// TwinCAT 3 PLC project Untitled1
// ProgramVersion: 3.1.4024.0
// libraries:
//   Tc2_Standard, * (Beckhoff Automation GmbH)
//   Tc2_System, * (Beckhoff Automation GmbH)
//   Tc3_Module, * (Beckhoff Automation GmbH)
// project tree:
//   DUTs/ KOMANDA.TcDUT (not stored), POZAYZ.TcDUT (not stored), POZICIJA.TcDUT (not stored), Valj.TcDUT (not stored)
//   GVLs/ AUTO.TcGVL, GVL.TcGVL (not stored)
//   / PlcTask.TcTTO (not stored)
//   POUs/ AutoMove.TcPOU (not stored), Counter.TcPOU (not stored), Init.TcPOU, MAIN.TcPOU (not stored), Motor.TcPOU (not stored), MotorControla.TcPOU, Multiplex.TcPOU (not stored), Automatic.TcPOU, AutoMove2.TcPOU, Test.TcPOU (not stored), TrackingLogic.TcPOU (not stored)
// real-time tasks:
//   TASK PlcTask: cycle T#10ms, priority 20, ADS port 350
// I/O:
//   DEVICE Device 1 (EtherCAT), AmsNetId 5.132.85.185.2.1
//     Term 1 (EK1200) [EK1200-7000 EtherCAT Power supply (1,5A E-Bus)]
//       Term 2 (EL1859) [EL1859 8Ch. Dig. Input 24V, 3ms, 8Ch. Dig. Output 24V, 0.5A]
//       Term 3 (EL1859) [EL1859 8Ch. Dig. Input 24V, 3ms, 8Ch. Dig. Output 24V, 0.5A]
//       Term 4 (EL5152) [EL5152 2Ch. Inc. Encoder]
//       Term 5 (EL9011) [EL9011 End Terminal]
//   DEVICE Device 2 (NOV-DP-RAM)
//   DEVICE Device 5 (CX7000), AmsNetId 5.132.85.185.6.1
//     Term 1 (CX7028) [CX7028-0000-0118]
//       modules: Module 1 (DIO_2x), Module 3 (DIO_2x), Module 5 (DI_2x), Module 7 (DI_2x)
// variable links:
//   Untitled1/Untitled1 Instance <-> Device 1 (EtherCAT)/Term 1 (EK1200)/Term 2 (EL1859)
//     PlcTask Inputs/GVL.KSD <-> Channel 5/Input
//     PlcTask Inputs/GVL.KSI <-> Channel 3/Input
//     PlcTask Inputs/GVL.KSP <-> Channel 7/Input
//     PlcTask Inputs/GVL.KSV <-> Channel 1/Input
//     PlcTask Inputs/GVL.StD <-> Channel 6/Input
//     PlcTask Inputs/GVL.StI <-> Channel 4/Input
//     PlcTask Inputs/GVL.StP <-> Channel 8/Input
//     PlcTask Inputs/GVL.StV <-> Channel 2/Input
//     PlcTask Outputs/GVL.MDP <-> Channel 14/Output
//     PlcTask Outputs/GVL.MDS <-> Channel 13/Output
//     PlcTask Outputs/GVL.MIP <-> Channel 12/Output
//     PlcTask Outputs/GVL.MIS <-> Channel 11/Output
//     PlcTask Outputs/GVL.MPP <-> Channel 16/Output
//     PlcTask Outputs/GVL.MPS <-> Channel 15/Output
//     PlcTask Outputs/GVL.MVP <-> Channel 10/Output
//     PlcTask Outputs/GVL.MVS <-> Channel 9/Output
//   Untitled1/Untitled1 Instance <-> Device 5 (CX7000)/Term 1 (CX7028)
//     PlcTask Inputs/GVL.GreenButton <-> Module 3 (DIO_2x)/DIO_2x Input Channel 2/Input
//     PlcTask Inputs/GVL.LLBButton <-> Module 5 (DI_2x)/DI_2x Input Channel 1/Input
//     PlcTask Inputs/GVL.LRBButton <-> Module 5 (DI_2x)/DI_2x Input Channel 2/Input
//     PlcTask Inputs/GVL.RedButton <-> Module 1 (DIO_2x)/DIO_2x Inputs Channel 1/Input
//     PlcTask Inputs/GVL.ToggleSwitch <-> Module 7 (DI_2x)/DI_2x Inputs Channel 1/Input
//     PlcTask Inputs/GVL.ULBButton <-> Module 1 (DIO_2x)/DIO_2x Inputs Channel 2/Input
//     PlcTask Inputs/GVL.URBButton <-> Module 3 (DIO_2x)/DIO_2x Input Channel 1/Input
//     PlcTask Outputs/GVL.LEDGreen <-> Module 3 (DIO_2x)/DIO_2x Outputs Channel 1/Output
//     PlcTask Outputs/GVL.LEDLBlue <-> Module 3 (DIO_2x)/DIO_2x Outputs Channel 2/Output
//     PlcTask Outputs/GVL.LEDRed <-> Module 1 (DIO_2x)/DIO_2x Outputs Channel 1/Output
//     PlcTask Outputs/GVL.LEDUBlue <-> Module 1 (DIO_2x)/DIO_2x Outputs Channel 2/Output

// ---- GVLs/AUTO.TcGVL
{attribute 'qualified_only'}
VAR_GLOBAL
	Varno :BOOL := FALSE;
	MotorIzbira : INT;
	VrtenjePremik : BOOL;
	VrtenjeSmer : BOOL;
	DvigPremik : BOOL;
	DvigSmer : BOOL;
	IztegPremik : BOOL;
	IztegSmer : BOOL;
	PrijemPremik : BOOL;
	PrijemSmer : BOOL;
	Current: POZICIJA;
	N: INT := 5; //v InstructionSize
	Komande0: ARRAY [0..4] OF POZICIJA := [(A := 0, Y := 0, Z := 0, P:= 0 ), 
		(A := 100, Y := 40, Z := 50, P:= 15 ),
		(A := 80, Y := 20, Z := 30, P:= 0 ),
		(A := 120, Y := 0, Z := 15, P:= 12 ),
		(A := 100, Y := 0, Z := 15, P:= 0 )];
	Status: INT := 0;
	PositionNum: INT := 2; // ne rabi
	ItemNumber : INT := 2; //ne rabi
	StageSelect : INT := 0;
	Recept : INT := 0;
	VRoki : INT := 0;
	Positions: ARRAY [1..11] OF POZAYZ := [
			(A := 30, Y:=60, Z:= 105),
			(A := 30, Y:=60, Z:= 62),
			(A := 30, Y:=60, Z:= 20),
			(A := 60, Y:=60, Z:= 105),
			(A := 60, Y:=60, Z:= 62), // 5
			(A := 50, Y:=60, Z:= 105),
			(A := 50, Y:=60, Z:= 62),
			(A := 37, Y:=60, Z:= 105),
			(A := 40, Y:=45, Z:= 105),
			(A := 43, Y:=60, Z:= 105),
			(A := 33, Y:=0, Z:= 50)]; // 10
	Items: ARRAY [1..5] OF POZAYZ := [
			(A := 5, Y:=60, Z:= 20),
			(A := 5, Y:=60, Z:= 62),
			(A := 5, Y:=60, Z:= 105),
			(A := 50, Y:=60, Z:= 105),
			(A := 50, Y:=60, Z:= 62)];
	StageMax : INT :=10;
	Stages :  ARRAY [1 .. 3] OF ARRAY [1 .. 9] OF KOMANDA :=  [[
		(I := 1, T := 0, P := 16),
		(I := 0, T := 1, P := 0),
		(I := 2, T := 0, P := 16),
		(I := 0, T := 2, P := 0),
		(I := 3, T := 0, P := 16), // 5
		(I := 0, T := 3, P := 0),
		(I := 2, T := 0, P := 16),
		(I := 0, T := 9, P := 0),
		(I := 0, T := 11, P := 0)],
[
		(I := 5, T := 0, P := 16),
		(I := 0, T := 4, P := 0),
		(I := 4, T := 0, P := 16),
		(I := 0, T := 5, P := 0),
		(I := 4, T := 0, P := 16), // 5
		(I := 0, T := 6, P := 0),
		(I := 5, T := 0, P := 16),
		(I := 0, T := 7, P := 0),
		(I := 0, T := 11, P := 0)],
[
		(I := 1, T := 0, P := 16),
		(I := 0, T := 10, P := 0),
		(I := 2, T := 0, P := 16),
		(I := 0, T := 8, P := 0),
		(I := 3, T := 0, P := 16), // 5
		(I := 0, T := 9, P := 0),
		(I := 2, T := 0, P := 16),
		(I := 0, T := 1, P := 0),
		(I := 0, T := 11, P := 0)]];
END_VAR

// ---- POUs/Init.TcPOU
FUNCTION_BLOCK Init
VAR_INPUT
END_VAR
VAR_OUTPUT
END_VAR
VAR
	isInit: BOOL := FALSE;
END_VAR

IF NOT isInit AND GVL.ToggleSwitch = FALSE THEN
	IF NOT GVL.KSV THEN
		AUTO.MotorIzbira := 1;
		AUTO.VrtenjeSmer := TRUE;
		AUTO.VrtenjePremik := TRUE;
	ELSIF NOT GVL.KSD THEN
		AUTO.VrtenjePremik:= FALSE;
		AUTO.MotorIzbira := 2;
		AUTO.DvigSmer := TRUE;
		AUTO.DvigPremik := TRUE;
	ELSIF NOT GVL.KSP THEN
		AUTO.MotorIzbira := 4;
		AUTO.PrijemSmer := TRUE;
		AUTO.PrijemPremik := TRUE;
	ELSE
		AUTO.MotorIzbira := 0;
		AUTO.Current.Y := 0;
		IF GVL.ULBButton = TRUE THEN
			AUTO.Recept := 1;
		ELSIF GVL.URBButton = TRUE THEN
			AUTO.Recept:= 2;
		ELSIF GVL.LLBButton= TRUE THEN
			AUTO.Recept := 3;
		END_IF
		IF AUTO.Recept <> 0 THEN
			AUTO.StageSelect := 1;
			isInit := TRUE;
		END_IF
		
	END_IF
END_IF

END_FUNCTION_BLOCK

// ---- POUs/MotorControla.TcPOU
FUNCTION_BLOCK MotorControla
VAR_INPUT
	Premik: BOOL;
	Smer: BOOL;
	Select: BOOL;
	KS: BOOL;
	Step: BOOL;
	Limes: WORD;
END_VAR
VAR_OUTPUT
	OutPremik: BOOL;
	OutSmer: BOOL;
	Interlock: BOOL;
	Stop: BOOL;
	Position: WORD;
END_VAR
VAR
	R_TRIG_0: R_TRIG;
	Dump: TIME;
	InL: TOF;
	RS_0: RS;

	R_TRIG_1: R_TRIG;
	TON0: TON;
	TON1: TON;
	TON_0: TON;
	Counter_0: Counter;
	F_TRIG_0: F_TRIG;
	InL1: TOF;
	IntL1: BOOL;
	IntL2: BOOL;
	IntL3: BOOL;
END_VAR
//dODAJ COLLISION DETECTION AND AVOIDANCE
//ZRIHTAJ SMER, KI SE SLABO SPREMINJA

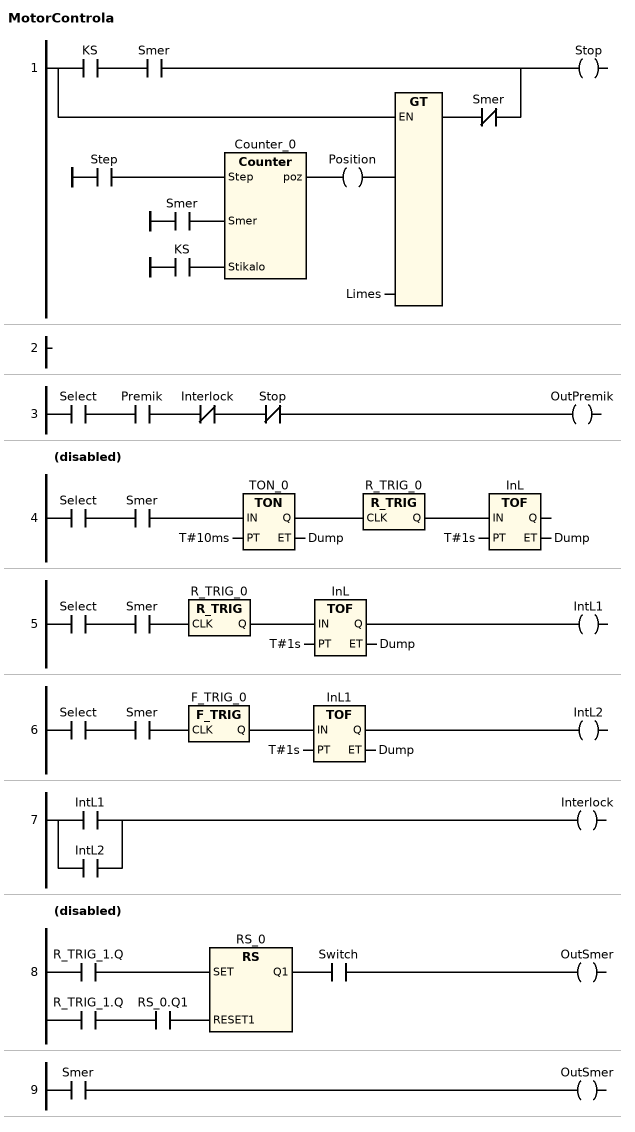
// NETWORK 1
Counter_0(Step := Step, Smer := Smer, Stikalo := KS); // Counter
Position := Counter_0.poz;
Stop := KS AND Smer OR Counter_0.poz > Limes AND NOT Smer;

// NETWORK 2

// NETWORK 3
OutPremik := Select AND Premik AND NOT Interlock AND NOT Stop;

// NETWORK 4 (disabled)
// TON_0(IN := Select AND Smer, PT := T#10ms, ET => Dump); // TON
// R_TRIG_0(CLK := TON_0.Q); // R_TRIG
// InL(IN := R_TRIG_0.Q, PT := T#1s, ET => Dump); // TOF

// NETWORK 5
R_TRIG_0(CLK := Select AND Smer); // R_TRIG
InL(IN := R_TRIG_0.Q, PT := T#1s, ET => Dump); // TOF
IntL1 := InL.Q;

// NETWORK 6
F_TRIG_0(CLK := Select AND Smer); // F_TRIG
InL1(IN := F_TRIG_0.Q, PT := T#1s, ET => Dump); // TOF
IntL2 := InL1.Q;

// NETWORK 7
Interlock := IntL1 OR IntL2;

// NETWORK 8 (disabled)
// RS_0(SET := R_TRIG_1.Q, RESET1 := R_TRIG_1.Q AND RS_0.Q1); // RS
// OutSmer := RS_0.Q1 AND Switch;

// NETWORK 9
OutSmer := Smer;

END_FUNCTION_BLOCK

// ---- POUs/Automatic.TcPOU
PROGRAM Automatic
VAR
	foo : BOOL;
	motor_1 : Motor;
	auto_move : AutoMove;
	auto_move_2 : AutoMove2;
	tracking : TrackingLogic;
	init : Init;
END_VAR


init();
auto_move_2();
motor_1();
tracking();

END_PROGRAM

// ---- POUs/AutoMove2.TcPOU
FUNCTION_BLOCK AutoMove2
VAR_INPUT
END_VAR
VAR_OUTPUT
END_VAR
VAR
	Target : POZAYZ;
END_VAR

IF AUTO.StageSelect > 0 AND AUTO.StageSelect < AUTO.StageMax THEN
	IF AUTO.Varno = FALSE THEN
		AUTO.MotorIzbira := 3;
		AUTO.IztegSmer := TRUE;
		AUTO.IztegPremik := TRUE;
		IF AUTO.Current.Y = 0 THEN
			AUTO.Varno := TRUE;
		END_IF
	ELSIF AUTO.Stages[AUTO.Recept][Auto.StageSelect].I = 0 THEN
		Target := AUTO.Positions[AUTO.Stages[AUTO.Recept][Auto.StageSelect].T];
		IF AUTO.Current.Z <> Target.Z  THEN
			AUTO.MotorIzbira := 2;
			IF AUTO.Current.Z > Target.Z THEN
				AUTO.DvigSmer := TRUE;
			ELSE
				AUTO.DvigSmer := FALSE;
			END_IF
		AUTO.DvigPremik := TRUE;
		ELSIF AUTO.Current.A <> Target.A  THEN
			AUTO.MotorIzbira := 1;
			IF AUTO.Current.A > Target.A THEN
				AUTO.VrtenjeSmer := TRUE;
			ELSE
				AUTO.VrtenjeSmer := FALSE;
			END_IF
			AUTO.VrtenjePremik := TRUE;
		ELSIF AUTO.Current.Y <> Target.Y  THEN
			AUTO.MotorIzbira := 3;
			IF AUTO.Current.Y > Target.Y THEN
				AUTO.IztegSmer := TRUE;
			ELSE
				AUTO.IztegSmer := FALSE;
			END_IF
			AUTO.IztegPremik := TRUE;
		ELSIF AUTO.Current.P <> AUTO.Stages[AUTO.Recept][Auto.StageSelect].P  THEN
			AUTO.MotorIzbira := 4;
			IF AUTO.Current.P > AUTO.Stages[AUTO.Recept][Auto.StageSelect].P THEN
				AUTO.PrijemSmer := TRUE;
			ELSE
				AUTO.PrijemSmer := FALSE;
			END_IF
			AUTO.PrijemPremik := TRUE;
		ELSE
			AUTO.VrtenjePremik := FALSE;
			AUTO.DvigPremik := FALSE;
			AUTO.IztegPremik := FALSE;
			AUTO.PrijemPremik := FALSE;
			AUTO.StageSelect := AUTO.StageSelect + 1;
			AUTO.Varno := FALSE;
		END_IF
	ELSE
		Target := AUTO.Items[AUTO.Stages[AUTO.Recept][Auto.StageSelect].I];
			IF AUTO.Current.A <> Target.A  THEN
			AUTO.MotorIzbira := 1;
			IF AUTO.Current.A > Target.A THEN
				AUTO.VrtenjeSmer := TRUE;
			ELSE
				AUTO.VrtenjeSmer := FALSE;
			END_IF
			AUTO.VrtenjePremik := TRUE;
		ELSIF AUTO.Current.Z <> Target.Z  THEN
			AUTO.MotorIzbira := 2;
			IF AUTO.Current.Z > Target.Z THEN
				AUTO.DvigSmer := TRUE;
			ELSE
				AUTO.DvigSmer := FALSE;
			END_IF
			AUTO.DvigPremik := TRUE;
		ELSIF AUTO.Current.Y <> Target.Y  THEN
			AUTO.MotorIzbira := 3;
			IF AUTO.Current.Y > Target.Y THEN
				AUTO.IztegSmer := TRUE;
			ELSE
				AUTO.IztegSmer := FALSE;
			END_IF
			AUTO.IztegPremik := TRUE;
		ELSIF AUTO.Current.P <> AUTO.Stages[AUTO.Recept][Auto.StageSelect].P  THEN
			AUTO.MotorIzbira := 4;
			IF AUTO.Current.P > AUTO.Stages[AUTO.Recept][Auto.StageSelect].P THEN
				AUTO.PrijemSmer := TRUE;
			ELSE
				AUTO.PrijemSmer := FALSE;
			END_IF
			AUTO.PrijemPremik := TRUE;
		ELSE
			AUTO.VrtenjePremik := FALSE;
			AUTO.DvigPremik := FALSE;
			AUTO.IztegPremik := FALSE;
			AUTO.PrijemPremik := FALSE;
			AUTO.StageSelect := AUTO.StageSelect + 1;
			IF AUTO.Recept = 2 AND AUTO.StageSelect = AUTO.StageMax THEN
				AUTO.StageSelect := 1;
			END_IF
			AUTO.Varno := FALSE;
		END_IF
	END_IF
	
END_IF

END_FUNCTION_BLOCK
